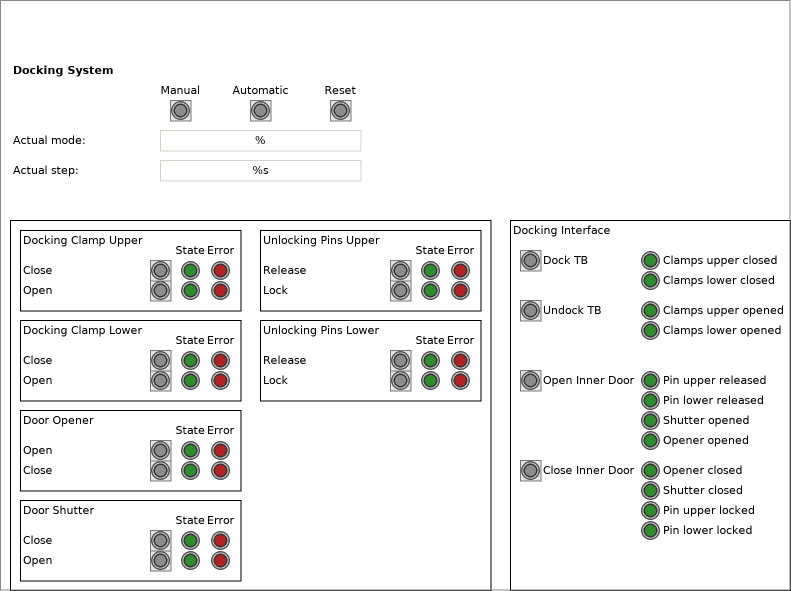
VISUALIZATION DockingInterface  // 791x591
    Rectangle (10,220 481x371)
    Rectangle (20,230 221x81)
    Lamp1 (180,260 21x21), variable: GVL_Modules.g_emDockingInterface.s_cmDockingClampsUpper.s_fbHmiLedIsOn.i_bStaLed, style: Lamp-Lamp1-Green
    Lamp1 (210,260 21x21), variable: GVL_Modules.g_emDockingInterface.s_cmDockingClampsUpper.s_fbHmiLedErrorOn.i_bStaLed, style: Lamp-Lamp1-Red
    PushSwitch (150,280 21x21), variable: GVL_Modules.g_emDockingInterface.s_cmDockingClampsUpper.s_fbHmiBtnManualOff.s_bFromHmiPressed, behaviour: TAP, style: Switch-PushSwitch-Gray
    PushSwitch (150,260 21x21), variable: GVL_Modules.g_emDockingInterface.s_cmDockingClampsUpper.s_fbHmiBtnManualOn.s_bFromHmiPressed, behaviour: TAP, style: Switch-PushSwitch-Gray
    Label (20,260 91x21), "Close"
    Label (20,280 78x21), "Open"
    Label (20,230 221x21), "Docking Clamp Upper"
    Lamp1 (180,280 21x21), variable: GVL_Modules.g_emDockingInterface.s_cmDockingClampsUpper.s_fbHmiLedIsOff.i_bStaLed, style: Lamp-Lamp1-Green
    Lamp1 (210,280 21x21), variable: GVL_Modules.g_emDockingInterface.s_cmDockingClampsUpper.s_fbHmiLedErrorOff.i_bStaLed, style: Lamp-Lamp1-Red
    Label (170,240 41x21), "State"
    Label (200,240 41x21), "Error"
    Rectangle (20,320 221x81)
    Lamp1 (180,350 21x21), variable: GVL_Modules.g_emDockingInterface.s_cmDockingClampsLower.s_fbHmiLedIsOn.i_bStaLed, style: Lamp-Lamp1-Green
    Lamp1 (210,350 21x21), variable: GVL_Modules.g_emDockingInterface.s_cmDockingClampsLower.s_fbHmiLedErrorOn.i_bStaLed, style: Lamp-Lamp1-Red
    PushSwitch (150,370 21x21), variable: GVL_Modules.g_emDockingInterface.s_cmDockingClampsLower.s_fbHmiBtnManualOff.s_bFromHmiPressed, behaviour: TAP, style: Switch-PushSwitch-Gray
    PushSwitch (150,350 21x21), variable: GVL_Modules.g_emDockingInterface.s_cmDockingClampsLower.s_fbHmiBtnManualOn.s_bFromHmiPressed, behaviour: TAP, style: Switch-PushSwitch-Gray
    Label (20,350 91x21), "Close"
    Label (20,370 78x21), "Open"
    Label (20,320 221x21), "Docking Clamp Lower"
    Lamp1 (180,370 21x21), variable: GVL_Modules.g_emDockingInterface.s_cmDockingClampsLower.s_fbHmiLedIsOff.i_bStaLed, style: Lamp-Lamp1-Green
    Lamp1 (210,370 21x21), variable: GVL_Modules.g_emDockingInterface.s_cmDockingClampsLower.s_fbHmiLedErrorOff.i_bStaLed, style: Lamp-Lamp1-Red
    Label (170,330 41x21), "State"
    Label (200,330 41x21), "Error"
    Rectangle (260,230 221x81)
    Lamp1 (420,260 21x21), variable: GVL_Modules.g_emDockingInterface.s_cmUnlockingPinUpper.s_fbHmiLedIsOn.i_bStaLed, style: Lamp-Lamp1-Green
    Lamp1 (450,260 21x21), variable: GVL_Modules.g_emDockingInterface.s_cmUnlockingPinUpper.s_fbHmiLedErrorOn.i_bStaLed, style: Lamp-Lamp1-Red
    PushSwitch (390,280 21x21), variable: GVL_Modules.g_emDockingInterface.s_cmUnlockingPinUpper.s_fbHmiBtnManualOff.s_bFromHmiPressed, behaviour: TAP, style: Switch-PushSwitch-Gray
    PushSwitch (390,260 21x21), variable: GVL_Modules.g_emDockingInterface.s_cmUnlockingPinUpper.s_fbHmiBtnManualOn.s_bFromHmiPressed, behaviour: TAP, style: Switch-PushSwitch-Gray
    Label (260,260 91x21), "Release"
    Label (260,280 78x21), "Lock"
    Label (260,230 221x21), "Unlocking Pins Upper"
    Lamp1 (420,280 21x21), variable: GVL_Modules.g_emDockingInterface.s_cmUnlockingPinUpper.s_fbHmiLedIsOff.i_bStaLed, style: Lamp-Lamp1-Green
    Lamp1 (450,280 21x21), variable: GVL_Modules.g_emDockingInterface.s_cmUnlockingPinUpper.s_fbHmiLedErrorOff.i_bStaLed, style: Lamp-Lamp1-Red
    Label (410,240 41x21), "State"
    Label (440,240 41x21), "Error"
    Rectangle (260,320 221x81)
    Lamp1 (420,350 21x21), variable: GVL_Modules.g_emDockingInterface.s_cmUnlockingPinLower.s_fbHmiLedIsOn.i_bStaLed, style: Lamp-Lamp1-Green
    Lamp1 (450,350 21x21), variable: GVL_Modules.g_emDockingInterface.s_cmUnlockingPinLower.s_fbHmiLedErrorOn.i_bStaLed, style: Lamp-Lamp1-Red
    PushSwitch (390,370 21x21), variable: GVL_Modules.g_emDockingInterface.s_cmUnlockingPinLower.s_fbHmiBtnManualOff.s_bFromHmiPressed, behaviour: TAP, style: Switch-PushSwitch-Gray
    PushSwitch (390,350 21x21), variable: GVL_Modules.g_emDockingInterface.s_cmUnlockingPinLower.s_fbHmiBtnManualOn.s_bFromHmiPressed, behaviour: TAP, style: Switch-PushSwitch-Gray
    Label (260,350 91x21), "Release"
    Label (260,370 78x21), "Lock"
    Label (260,320 221x21), "Unlocking Pins Lower"
    Lamp1 (420,370 21x21), variable: GVL_Modules.g_emDockingInterface.s_cmUnlockingPinLower.s_fbHmiLedIsOff.i_bStaLed, style: Lamp-Lamp1-Green
    Lamp1 (450,370 21x21), variable: GVL_Modules.g_emDockingInterface.s_cmUnlockingPinLower.s_fbHmiLedErrorOff.i_bStaLed, style: Lamp-Lamp1-Red
    Label (410,330 41x21), "State"
    Label (440,330 41x21), "Error"
    Rectangle (20,410 221x81)
    Lamp1 (180,440 21x21), variable: GVL_Modules.g_emDockingInterface.s_cmDoorOpener.s_fbHmiLedIsOn.i_bStaLed, style: Lamp-Lamp1-Green
    Lamp1 (210,440 21x21), variable: GVL_Modules.g_emDockingInterface.s_cmDoorOpener.s_fbHmiLedErrorOn.i_bStaLed, style: Lamp-Lamp1-Red
    PushSwitch (150,460 21x21), variable: GVL_Modules.g_emDockingInterface.s_cmDoorOpener.s_fbHmiBtnManualOff.s_bFromHmiPressed, behaviour: TAP, style: Switch-PushSwitch-Gray
    PushSwitch (150,440 21x21), variable: GVL_Modules.g_emDockingInterface.s_cmDoorOpener.s_fbHmiBtnManualOn.s_bFromHmiPressed, behaviour: TAP, style: Switch-PushSwitch-Gray
    Label (20,440 91x21), "Open"
    Label (20,460 78x21), "Close"
    Label (20,410 221x21), "Door Opener"
    Lamp1 (180,460 21x21), variable: GVL_Modules.g_emDockingInterface.s_cmDoorOpener.s_fbHmiLedIsOff.i_bStaLed, style: Lamp-Lamp1-Green
    Lamp1 (210,460 21x21), variable: GVL_Modules.g_emDockingInterface.s_cmDoorOpener.s_fbHmiLedErrorOff.i_bStaLed, style: Lamp-Lamp1-Red
    Label (170,420 41x21), "State"
    Label (200,420 41x21), "Error"
    Rectangle (20,500 221x81)
    Lamp1 (180,530 21x21), variable: GVL_Modules.g_emDockingInterface.s_cmDoorShutter.s_fbHmiLedIsOn.i_bStaLed, style: Lamp-Lamp1-Green
    Lamp1 (210,530 21x21), variable: GVL_Modules.g_emDockingInterface.s_cmDoorShutter.s_fbHmiLedErrorOn.i_bStaLed, style: Lamp-Lamp1-Red
    PushSwitch (150,550 21x21), variable: GVL_Modules.g_emDockingInterface.s_cmDoorShutter.s_fbHmiBtnManualOff.s_bFromHmiPressed, behaviour: TAP, style: Switch-PushSwitch-Gray
    PushSwitch (150,530 21x21), variable: GVL_Modules.g_emDockingInterface.s_cmDoorShutter.s_fbHmiBtnManualOn.s_bFromHmiPressed, behaviour: TAP, style: Switch-PushSwitch-Gray
    Label (20,530 91x21), "Close"
    Label (20,550 78x21), "Open"
    Label (20,500 221x21), "Door Shutter"
    Lamp1 (180,550 21x21), variable: GVL_Modules.g_emDockingInterface.s_cmDoorShutter.s_fbHmiLedIsOff.i_bStaLed, style: Lamp-Lamp1-Green
    Lamp1 (210,550 21x21), variable: GVL_Modules.g_emDockingInterface.s_cmDoorShutter.s_fbHmiLedErrorOff.i_bStaLed, style: Lamp-Lamp1-Red
    Label (170,510 41x21), "State"
    Label (200,510 41x21), "Error"
    Label (10,160 71x21), "Actual step:"
    PushSwitch (330,100 21x21), variable: GVL.g_unCleanroomConnect.s_fbHmiBtnReset.s_bFromHmiPressed, behaviour: TAP, style: Switch-PushSwitch-Gray
    Rectangle (510,220 281x371)
    PushSwitch (520,300 21x21), variable: GVL_Modules.g_emDockingInterface.s_fbHmiBtnUndockTB.s_bFromHmiPressed, behaviour: TAP, style: Switch-PushSwitch-Gray
    PushSwitch (520,250 21x21), variable: GVL_Modules.g_emDockingInterface.s_fbHmiBtnDockTB.s_bFromHmiPressed, behaviour: TAP, style: Switch-PushSwitch-Gray
    Label (540,250 101x21), "Dock TB"
    Label (540,300 101x21), "Undock TB"
    Label (510,220 221x21), "Docking Interface"
    PushSwitch (520,460 21x21), variable: GVL_Modules.g_emDockingInterface.s_fbHmiBtnCloseInnerDoor.s_bFromHmiPressed, behaviour: TAP, style: Switch-PushSwitch-Gray
    PushSwitch (520,370 21x21), variable: GVL_Modules.g_emDockingInterface.s_fbHmiBtnOpenInnerDoor.s_bFromHmiPressed, behaviour: TAP, style: Switch-PushSwitch-Gray
    Label (540,370 101x21), "Open Inner Door"
    Label (540,460 101x21), "Close Inner Door"
    Lamp1 (640,250 21x21), variable: GVL_Modules.g_emDockingInterface.s_cmDockingClampsUpper.s_fbHmiLedIsOn.i_bStaLed, style: Lamp-Lamp1-Green
    Lamp1 (640,270 21x21), variable: GVL_Modules.g_emDockingInterface.s_cmDockingClampsLower.s_fbHmiLedIsOn.i_bStaLed, style: Lamp-Lamp1-Green
    Lamp1 (640,300 21x21), variable: GVL_Modules.g_emDockingInterface.s_cmDockingClampsUpper.s_fbHmiLedIsOff.i_bStaLed, style: Lamp-Lamp1-Green
    Lamp1 (640,320 21x21), variable: GVL_Modules.g_emDockingInterface.s_cmDockingClampsLower.s_fbHmiLedIsOff.i_bStaLed, style: Lamp-Lamp1-Green
    Lamp1 (640,370 21x21), variable: GVL_Modules.g_emDockingInterface.s_cmUnlockingPinUpper.s_fbHmiLedIsOn.i_bStaLed, style: Lamp-Lamp1-Green
    Lamp1 (640,390 21x21), variable: GVL_Modules.g_emDockingInterface.s_cmUnlockingPinLower.s_fbHmiLedIsOn.i_bStaLed, style: Lamp-Lamp1-Green
    Lamp1 (640,410 21x21), variable: GVL_Modules.g_emDockingInterface.s_cmDoorShutter.s_fbHmiLedIsOff.i_bStaLed, style: Lamp-Lamp1-Green
    Lamp1 (640,430 21x21), variable: GVL_Modules.g_emDockingInterface.s_cmDoorOpener.s_fbHmiLedIsOn.i_bStaLed, style: Lamp-Lamp1-Green
    Label (660,430 131x21), "Opener opened"
    Label (660,410 131x21), "Shutter opened"
    Label (660,390 131x21), "Pin lower released"
    Label (660,370 131x21), "Pin upper released"
    Label (660,320 131x21), "Clamps lower opened"
    Label (660,300 131x21), "Clamps upper opened"
    Label (660,270 131x21), "Clamps lower closed"
    Label (660,250 131x21), "Clamps upper closed"
    Label (660,460 131x21), "Opener closed"
    Label (660,480 131x21), "Shutter closed"
    Label (660,520 131x21), "Pin lower locked"
    Label (660,500 131x21), "Pin upper locked"
    Lamp1 (640,500 21x21), variable: GVL_Modules.g_emDockingInterface.s_cmUnlockingPinUpper.s_fbHmiLedIsOff.i_bStaLed, style: Lamp-Lamp1-Green
    Lamp1 (640,520 21x21), variable: GVL_Modules.g_emDockingInterface.s_cmUnlockingPinLower.s_fbHmiLedIsOff.i_bStaLed, style: Lamp-Lamp1-Green
    Lamp1 (640,460 21x21), variable: GVL_Modules.g_emDockingInterface.s_cmDoorOpener.s_fbHmiLedIsOff.i_bStaLed, style: Lamp-Lamp1-Green
    Lamp1 (640,480 21x21), variable: GVL_Modules.g_emDockingInterface.s_cmDoorShutter.s_fbHmiLedIsOn.i_bStaLed, style: Lamp-Lamp1-Green
    Textfield (160,160 201x21), "%s", text variable: GVL_Modules.g_emDockingInterface.s_fbSeqDockingInterfaceControl.i_sStepName
    Label (320,80 41x21), "Reset"
    Label (10,130 71x21), "Actual mode:"
    Textfield (160,130 201x21), "%", text list: 'E_MODE', text index: GVL_Modules.g_emDockingInterface.i_eCtrlMode
    PushSwitch (170,100 21x21), variable: GVL.g_unCleanroomConnect.s_fbHmiBtnManual.s_bFromHmiPressed, behaviour: TAP, style: Switch-PushSwitch-Gray
    PushSwitch (250,100 21x21), variable: GVL.g_unCleanroomConnect.s_fbHmiBtnAutomatic.s_bFromHmiPressed, behaviour: TAP, style: Switch-PushSwitch-Gray
    Label (140,80 81x21), "Manual"
    Label (220,80 81x21), "Automatic"
    Label (10,60 141x21), "Docking System"
END_VISUALIZATION

(* stored: Version 1.1.0.1, ProductVersion 3.1.4024.12
   Visu DockingInterface: Id {67f9a1b9-3dca-44e0-8245-e665cd9ce16d} *)
